SUBAPPLICATION mapping_Uebung_033_VV_FORTE_PC_B (* LED Strip Blinkende LED *)
  (* Standard: 61499-2; Description: Copyright (c) 2023 HR Agrartechnik GmbH This program and the accompanying materials are made available under the terms of the Eclipse Public License 2.0 which is available at https://www.eclipse.org/legal/epl-2.0/ SPDX-License-Identifier: EPL-2.0 *)
  (* Version 1.0, 2023-10-23, Franz Höpfinger, HR Agrartechnik GmbH *)
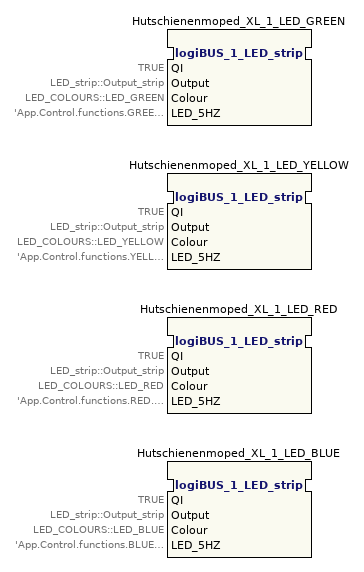
  FBS
    Hutschienenmoped_XL_1_LED_RED : logiBUS_1_LED_strip(QI := TRUE, Output := LED_strip::Output_strip, Colour := LED_COLOURS::LED_RED, LED_5HZ := 'App.Control.functions.RED.LED');
    Hutschienenmoped_XL_1_LED_GREEN : logiBUS_1_LED_strip(QI := TRUE, Output := LED_strip::Output_strip, Colour := LED_COLOURS::LED_GREEN, LED_5HZ := 'App.Control.functions.GREEN.LED');
    Hutschienenmoped_XL_1_LED_BLUE : logiBUS_1_LED_strip(QI := TRUE, Output := LED_strip::Output_strip, Colour := LED_COLOURS::LED_BLUE, LED_5HZ := 'App.Control.functions.BLUE.LED');
    Hutschienenmoped_XL_1_LED_YELLOW : logiBUS_1_LED_strip(QI := TRUE, Output := LED_strip::Output_strip, Colour := LED_COLOURS::LED_YELLOW, LED_5HZ := 'App.Control.functions.YELLOW.LED');
  END_FBS
END_SUBAPPLICATION
